// Gets the lower bound index of the array of specified type.
FUNCTION F_GetUDIntArrayLowerBound : T_Position // The lower bound index of the specified array.
VAR_IN_OUT
	arArray : ARRAY[*] OF UDINT; // The array to query.
END_VAR

F_GetUDIntArrayLowerBound := LOWER_BOUND(arArray, 1);

END_FUNCTION

(* stored: Version 1.1.0.1
   POU F_GetUDIntArrayLowerBound: Id {746cc107-cd14-0b90-0f46-0010227e1fa9}, SpecialFunc None *)
